FUNCTION_BLOCK Q_SetAudioVolume (* Command SetAudioVolume. *)
  (* Standard: ISO 11783-6; Description: Copyright (c) 2022 HR Agrartechnik GmbH This program and the accompanying materials are made available under the terms of the Eclipse Public License 2.0 which is available at https://www.eclipse.org/legal/epl-2.0/ SPDX-License-Identifier: EPL-2.0 see Description Tab *)
  (* Version 1.0, 2022-07-08, Franz Höpfinger, HR Agrartechnik GmbH *)
  (* Documentation:
  Command SetAudioVolume
   This command can be used to control the audio on the VT (volume) ( Part 6 - F.12 )
   param[in] {volume_percent, uint8_t}
   Volume 0 - 100 (%)
   Return Values: 
   int16_t
    - VT_E_NO_ERR (0) - OK
   - VT_E_OVERFLOW (-6) - buffer overflow
   - VT_E_NOACT (-8) - Command not possible in current state
   - VT_E_NO_INSTANCE (-21) - No VT client available
   - VT_E_ISO_INSTANCE_INVALID (-129) - Identifier for instance (connection) invalid
   - VT_E_HANDLE_INVALID (-128) - ErrorCause: invalid Handle
   - VT_E_NOT_ALIVE (-130) - Identifier for instance valid, but VT Dead.
  *)
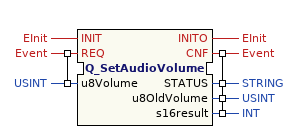
  EVENT_INPUT
    INIT : EInit; (* Service Initialization *)
    REQ WITH u8Volume; (* Service Request *)
  END_EVENT
  EVENT_OUTPUT
    INITO : EInit; (* Initialization Confirm *)
    CNF WITH STATUS, s16result, u8OldVolume; (* Confirmation of Requested Service *)
  END_EVENT
  VAR_INPUT
    u8Volume : USINT; (* Volume 0 - 100 (%) *)
  END_VAR
  VAR_OUTPUT
    STATUS : STRING; (* Service Status *)
    u8OldVolume : USINT; (* Old volume 0 - 100 (%) *)
    s16result : INT; (* retval see description *)
  END_VAR
END_FUNCTION_BLOCK
